// TIA Portal V19 program export: 4 tag tables, 0 data types, 0 data blocks, 3 code blocks (in call order from the OBs), 5 instance data blocks

VAR_GLOBAL   // PLC tag table "Alarm_Tags"
   ACKPB AT %M3.3 : Bool;   // Alarm ACK
   RESETPB AT %M3.4 : Bool;   // Alarm Reset
   Alarm_1 AT %M3.5 : Bool;   // Alarm #No1
   Alarm1ACKED AT %M3.6 : Bool;   // Alarm #1 Acknowledged
   Alarm1LED AT %M3.7 : Bool;   // Alarm #1 LED
   StopBelt AT %M4.0 : Bool;   // E-Stop The Belt
   Alarm_2 AT %M4.1 : Bool;   // Alarm #No2
   Alarm2ACKED AT %M4.2 : Bool;   // Alarm #2 Acknowledged
   Alarm2LED AT %M4.3 : Bool;   // Alarm #2 LED
END_VAR

VAR_GLOBAL   // PLC tag table "Clock_Tags"
   Clock_Byte AT %MB0 : Byte;
   Clock_10Hz AT %M0.0 : Bool;
   Clock_5Hz AT %M0.1 : Bool;
   "Clock_2.5Hz" AT %M0.2 : Bool;
   Clock_2Hz AT %M0.3 : Bool;
   "Clock_1.25Hz" AT %M0.4 : Bool;
   Clock_1Hz AT %M0.5 : Bool;
   "Clock_0.625Hz" AT %M0.6 : Bool;
   "Clock_0.5Hz" AT %M0.7 : Bool;
END_VAR

VAR_GLOBAL   // PLC tag table "Level_Tags"
   Pump1_Mode AT %M5.1 : Bool;   // Running Mode ( Auto or Manual)
   Pump1_Start_Manual AT %M5.2 : Bool;   // Start Manual Mode
   Pump1_Stop_Manual AT %M5.3 : Bool;   // Stop Manual Mode
   Pump1_Start_Auto AT %M5.4 : Bool;   // Start Auto Mode
   Pump1_Stop_Auto AT %M5.5 : Bool;   // Stop Auto Mode
   Level_High AT %M5.6 : Bool;   // High Level Reached
   Level_Low AT %M5.7 : Bool;   // Low Level Reached
   Timer_Setting_Run AT %MD6 : DInt;   // Timer Settings for Running
   Pump1_Overload AT %M10.0 : Bool;   // Pump Overloaded
   Pump1_Reset_Fault AT %M10.1 : Bool;   // Pump Reset Fault
   Pump1 AT %Q0.0 : Bool;   // Pump 1 - Output
   Pump1_Fault AT %M10.2 : Bool;   // Pump 1 Fault Status
   Pump1_Run_Auto_Activated AT %M10.3 : Bool;   // Pump 1 Running in Auto
   Level_Meter AT %MW12 : Int;   // Level Meter Reading
   Sensor_Real AT %QD2 : Real;   // Real Sensor Reading ( Tank Level)
   High_SP AT %MD14 : Real;   // High Setpoint
   Low_SP AT %MD18 : Real;   // Low Setpoint
END_VAR

VAR_GLOBAL   // PLC tag table "Mixer_Tags"
   Mixer_Start_PB AT %M4.5 : Bool;   // Starts Mixer
   Mixer_Stop_PB AT %M4.6 : Bool;   // Stops Mixer
   Mixer_Hold AT %M4.7 : Bool;   // Mixer held In Running
   Mixer AT %M5.0 : Bool;   // Mixer Status
   "2Hz_Mixer" AT %M4.4 : Bool;   // 2HZ Signal
END_VAR

ORGANIZATION_BLOCK "Main"   // OB1, LAD, ProgramCycle
TITLE = "Main Program Sweep (Cycle)"
{ S7_Optimized_Access := 'TRUE' }
// stored: SetENOAutomatically false
   VAR_INPUT
      Initial_Call : Bool;   // Initial call of this OB
      Remanence : Bool;   // =True, if remanent data are available
   END_VAR
BEGIN

REGION Network 1: Dispenser
   // Running Code - Dispenser Project
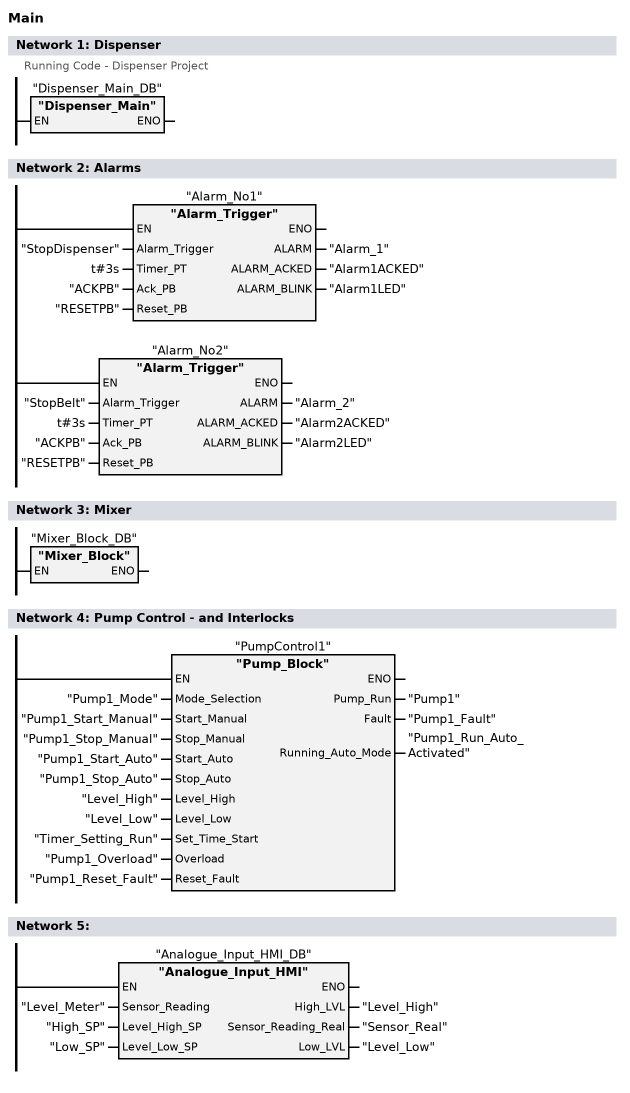
   RUNG wire#powerrail
      "Dispenser_Main_DB"()
   END_RUNG
   // the same network as SCL:
   "Dispenser_Main_DB"();   // "Dispenser_Main"
END_REGION

REGION Network 2: Alarms
   RUNG wire#powerrail
      "Alarm_No1"(Alarm_Trigger := "StopDispenser", Timer_PT := t#3s, Ack_PB := "ACKPB", Reset_PB := "RESETPB", ALARM => "Alarm_1", ALARM_ACKED => "Alarm1ACKED", ALARM_BLINK => "Alarm1LED")
   END_RUNG
   RUNG wire#powerrail
      "Alarm_No2"(Alarm_Trigger := "StopBelt", Timer_PT := t#3s, Ack_PB := "ACKPB", Reset_PB := "RESETPB", ALARM => "Alarm_2", ALARM_ACKED => "Alarm2ACKED", ALARM_BLINK => "Alarm2LED")
   END_RUNG
   // the same network as SCL:
   "Alarm_No1"(Alarm_Trigger := "StopDispenser",   // "Alarm_Trigger"
               Timer_PT := t#3s,
               Ack_PB := "ACKPB",
               Reset_PB := "RESETPB",
               ALARM => "Alarm_1",
               ALARM_ACKED => "Alarm1ACKED",
               ALARM_BLINK => "Alarm1LED");
   "Alarm_No2"(Alarm_Trigger := "StopBelt",   // "Alarm_Trigger"
               Timer_PT := t#3s,
               Ack_PB := "ACKPB",
               Reset_PB := "RESETPB",
               ALARM => "Alarm_2",
               ALARM_ACKED => "Alarm2ACKED",
               ALARM_BLINK => "Alarm2LED");
END_REGION

REGION Network 3: Mixer
   RUNG wire#powerrail
      "Mixer_Block_DB"()
   END_RUNG
   // the same network as SCL:
   "Mixer_Block_DB"();   // "Mixer_Block"
END_REGION

REGION Network 4: Pump Control - and Interlocks
   RUNG wire#powerrail
      "PumpControl1"(Mode_Selection := "Pump1_Mode", Start_Manual := "Pump1_Start_Manual", Stop_Manual := "Pump1_Stop_Manual", Start_Auto := "Pump1_Start_Auto", Stop_Auto := "Pump1_Stop_Auto", Level_High := "Level_High", Level_Low := "Level_Low", Set_Time_Start := "Timer_Setting_Run", Overload := "Pump1_Overload", Reset_Fault := "Pump1_Reset_Fault", Pump_Run => "Pump1", Fault => "Pump1_Fault", Running_Auto_Mode => "Pump1_Run_Auto_Activated")
   END_RUNG
   // the same network as SCL:
   "PumpControl1"(Mode_Selection := "Pump1_Mode",   // "Pump_Block"
                  Start_Manual := "Pump1_Start_Manual",
                  Stop_Manual := "Pump1_Stop_Manual",
                  Start_Auto := "Pump1_Start_Auto",
                  Stop_Auto := "Pump1_Stop_Auto",
                  Level_High := "Level_High",
                  Level_Low := "Level_Low",
                  Set_Time_Start := "Timer_Setting_Run",
                  Overload := "Pump1_Overload",
                  Reset_Fault := "Pump1_Reset_Fault",
                  Pump_Run => "Pump1",
                  Fault => "Pump1_Fault",
                  Running_Auto_Mode => "Pump1_Run_Auto_Activated");
END_REGION

REGION Network 5
   RUNG wire#powerrail
      "Analogue_Input_HMI_DB"(Sensor_Reading := "Level_Meter", Level_High_SP := "High_SP", Level_Low_SP := "Low_SP", High_LVL => "Level_High", Sensor_Reading_Real => "Sensor_Real", Low_LVL => "Level_Low")
   END_RUNG
   // the same network as SCL:
   "Analogue_Input_HMI_DB"(Sensor_Reading := "Level_Meter",   // "Analogue_Input_HMI"
                           Level_High_SP := "High_SP",
                           Level_Low_SP := "Low_SP",
                           High_LVL => "Level_High",
                           Sensor_Reading_Real => "Sensor_Real",
                           Low_LVL => "Level_Low");
END_REGION
END_ORGANIZATION_BLOCK

FUNCTION_BLOCK "Dispenser_Main"   // FB1, LAD
TITLE = Main Block for Dispenser Element and Conveyor Running
{ S7_Optimized_Access := 'TRUE' }
// Holds Code for Dispenser Project , Light Gates and Conveyor Belt Motor.
// stored: MemoryReserve 100, SetENOAutomatically false
   VAR_TEMP   // added for the SCL form of the ladder/FBD networks
      _w1 : Bool;
   END_VAR
BEGIN

REGION Network 1: Power Up
   // Enabled Power To System
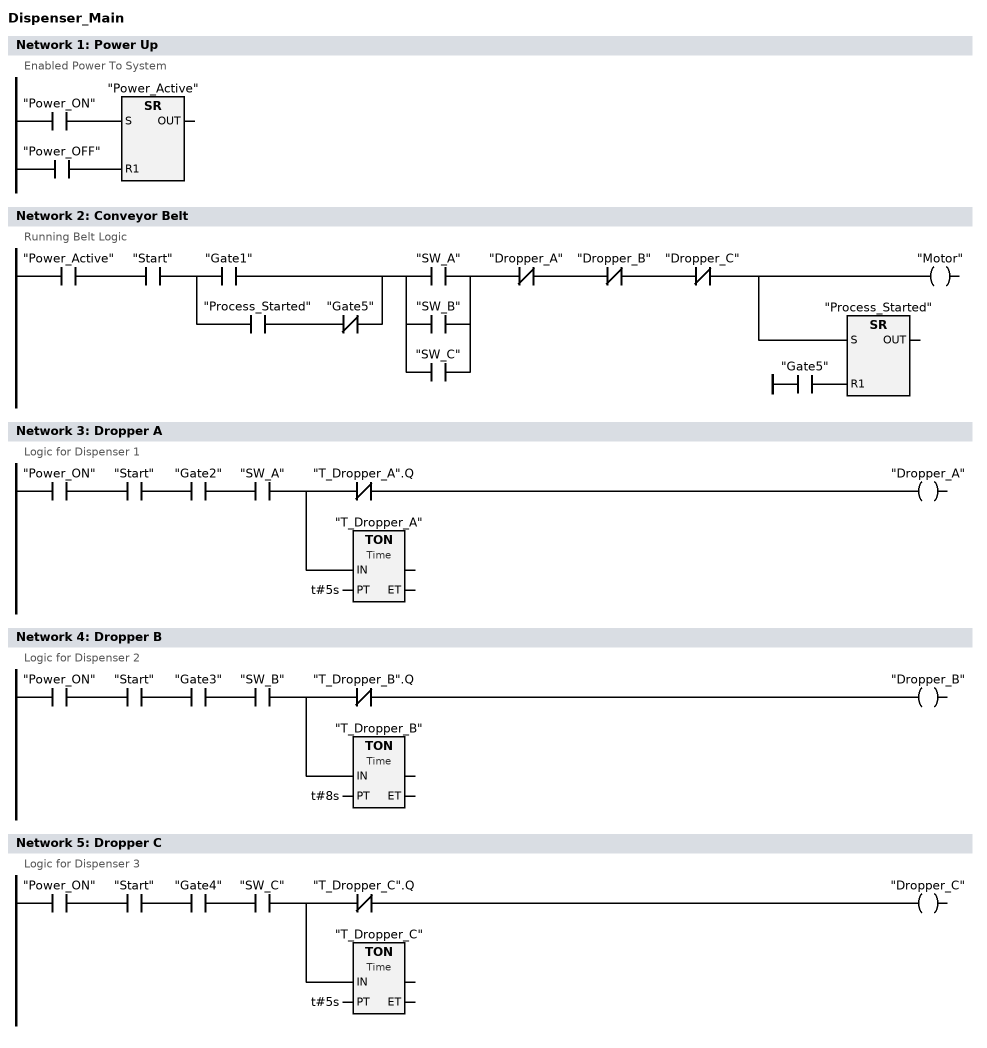
   RUNG wire#powerrail
      Contact( "Power_ON" )
      S_SR(operand := "Power_Active", r1 := wire#w1)
   END_RUNG
   RUNG wire#powerrail
      Contact( "Power_OFF" )
   END_RUNG wire#w1
   // the same network as SCL:
   IF "Power_ON" THEN
       "Power_Active" := TRUE;   // SR flip-flop
   END_IF;
   IF "Power_OFF" THEN "Power_Active" := FALSE; END_IF;
END_REGION

REGION Network 2: Conveyor Belt
   // Running Belt Logic
   RUNG wire#powerrail
      Contact( "Power_Active" )
      Contact( "Start" )
      wire#w1
      Contact( "Gate1" )
      wire#w2
      Contact( "SW_A" )
      wire#w3
      I_Contact( "Dropper_A" )
      I_Contact( "Dropper_B" )
      I_Contact( "Dropper_C" )
      wire#w4
      Coil( "Motor" )
   END_RUNG
   RUNG wire#w1
      Contact( "Process_Started" )
      I_Contact( "Gate5" )
   END_RUNG wire#w2
   RUNG wire#w2
      Contact( "SW_B" )
   END_RUNG wire#w3
   RUNG wire#w2
      Contact( "SW_C" )
   END_RUNG wire#w3
   RUNG wire#w4
      S_SR(operand := "Process_Started", r1 := wire#w5)
   END_RUNG
   RUNG wire#powerrail
      Contact( "Gate5" )
   END_RUNG wire#w5
   // the same network as SCL:
   "Motor" := "Power_Active" AND "Start" AND ("Gate1" OR ("Process_Started" AND NOT "Gate5")) AND ("SW_A" OR "SW_B" OR "SW_C") AND NOT "Dropper_A" AND NOT "Dropper_B" AND NOT "Dropper_C";
   IF "Motor" THEN
       "Process_Started" := TRUE;   // SR flip-flop
   END_IF;
   IF "Gate5" THEN "Process_Started" := FALSE; END_IF;
END_REGION

REGION Network 3: Dropper A
   // Logic for Dispenser 1
   RUNG wire#powerrail
      Contact( "Power_ON" )
      Contact( "Start" )
      Contact( "Gate2" )
      Contact( "SW_A" )
      wire#w1
      I_Contact( "T_Dropper_A".Q )
      Coil( "Dropper_A" )
   END_RUNG
   RUNG wire#w1
      { S7_Templates := "time_type := Time" } "T_Dropper_A".TON(pt := t#5s, et =>)
   END_RUNG
   // the same network as SCL:
   #_w1 := "Power_ON" AND "Start" AND "Gate2" AND "SW_A";
   "Dropper_A" := #_w1 AND NOT "T_Dropper_A".Q;
   "T_Dropper_A".TON(IN := #_w1, PT := t#5s);
END_REGION

REGION Network 4: Dropper B
   // Logic for Dispenser 2
   RUNG wire#powerrail
      Contact( "Power_ON" )
      Contact( "Start" )
      Contact( "Gate3" )
      Contact( "SW_B" )
      wire#w1
      I_Contact( "T_Dropper_B".Q )
      Coil( "Dropper_B" )
   END_RUNG
   RUNG wire#w1
      { S7_Templates := "time_type := Time" } "T_Dropper_B".TON(pt := t#8s, et =>)
   END_RUNG
   // the same network as SCL:
   #_w1 := "Power_ON" AND "Start" AND "Gate3" AND "SW_B";
   "Dropper_B" := #_w1 AND NOT "T_Dropper_B".Q;
   "T_Dropper_B".TON(IN := #_w1, PT := t#8s);
END_REGION

REGION Network 5: Dropper C
   // Logic for Dispenser 3
   RUNG wire#powerrail
      Contact( "Power_ON" )
      Contact( "Start" )
      Contact( "Gate4" )
      Contact( "SW_C" )
      wire#w1
      I_Contact( "T_Dropper_C".Q )
      Coil( "Dropper_C" )
   END_RUNG
   RUNG wire#w1
      { S7_Templates := "time_type := Time" } "T_Dropper_C".TON(pt := t#5s, et =>)
   END_RUNG
   // the same network as SCL:
   #_w1 := "Power_ON" AND "Start" AND "Gate4" AND "SW_C";
   "Dropper_C" := #_w1 AND NOT "T_Dropper_C".Q;
   "T_Dropper_C".TON(IN := #_w1, PT := t#5s);
END_REGION

REGION Network 6: Spare Network
END_REGION
END_FUNCTION_BLOCK

FUNCTION_BLOCK "Mixer_Block"   // FB3, LAD
TITLE = Control of Mixer Unit
{ S7_Optimized_Access := 'TRUE' }
// Simple Mixer Design and Animation
// stored: MemoryReserve 100, SetENOAutomatically false
BEGIN

REGION Network 1: Start Mixer
   // Turns Mixer On , Refreshes at 2Hz for Animation.
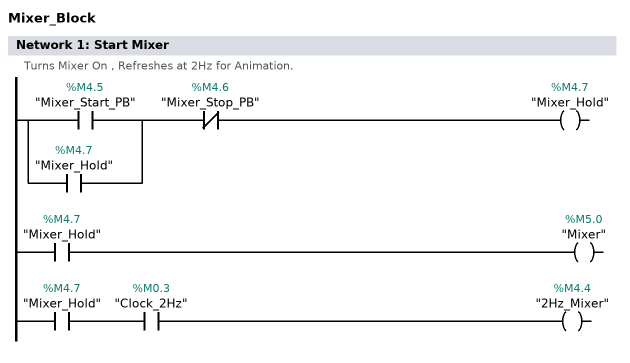
   RUNG wire#powerrail
      Contact( "Mixer_Start_PB" )
      wire#w1
      I_Contact( "Mixer_Stop_PB" )
      Coil( "Mixer_Hold" )
   END_RUNG
   RUNG wire#powerrail
      Contact( "Mixer_Hold" )
   END_RUNG wire#w1
   RUNG wire#powerrail
      Contact( "Mixer_Hold" )
      Coil( "Mixer" )
   END_RUNG
   RUNG wire#powerrail
      Contact( "Mixer_Hold" )
      Contact( "Clock_2Hz" )
      Coil( "2Hz_Mixer" )
   END_RUNG
   // the same network as SCL:
   "Mixer_Hold" := ("Mixer_Start_PB" OR "Mixer_Hold") AND NOT "Mixer_Stop_PB";
   "Mixer" := "Mixer_Hold";
   "2Hz_Mixer" := "Mixer_Hold" AND "Clock_2Hz";
END_REGION
END_FUNCTION_BLOCK

DATA_BLOCK "Alarm_No2"   // DB7
// stored: InstanceOfName Alarm_Trigger, InstanceOfType FB
"Alarm_Trigger"
   // VAR_INPUT
   //    Alarm_Trigger : Bool;
   //    Timer_PT : Time;
   //    Ack_PB : Bool;
   //    Reset_PB : Bool;
   // END_VAR
   // VAR_OUTPUT
   //    ALARM : Bool;
   //    ALARM_ACKED : Bool;
   //    ALARM_BLINK : Bool;
   // END_VAR
   // VAR
   //    Alarm_TD : Bool;
   //    Alarm_Active : Bool;
   //    Alarm_ACK : Bool;
   //    Alarm_Reset : Bool;
   //    Alarm_Timer { S7_SetPoint := 'True'} : TON_TIME;
   // END_VAR
BEGIN
END_DATA_BLOCK

DATA_BLOCK "Analogue_Input_HMI_DB"   // DB10
// stored: InstanceOfName Analogue_Input_HMI, InstanceOfType FB
"Analogue_Input_HMI"
   // VAR_INPUT
   //    Sensor_Reading { ExternalAccessible := 'False'; ExternalVisible := 'False'; ExternalWritable := 'False'} : Int;
   // END_VAR
   // VAR_OUTPUT
   //    High_LVL { ExternalAccessible := 'False'; ExternalVisible := 'False'; ExternalWritable := 'False'} : Bool;
   //    Sensor_Reading_Real { ExternalAccessible := 'False'; ExternalVisible := 'False'; ExternalWritable := 'False'} : Real;
   //    Low_LVL { ExternalAccessible := 'False'; ExternalVisible := 'False'; ExternalWritable := 'False'} : Bool;
   // END_VAR
   // VAR_IN_OUT
   //    Level_High_SP { ExternalAccessible := 'False'; ExternalVisible := 'False'; ExternalWritable := 'False'} : Real;
   //    Level_Low_SP { ExternalAccessible := 'False'; ExternalVisible := 'False'; ExternalWritable := 'False'} : Real;
   // END_VAR
BEGIN
END_DATA_BLOCK

DATA_BLOCK "Dispenser_Main_DB"   // DB4
// stored: InstanceOfName Dispenser_Main, InstanceOfType FB
"Dispenser_Main"
BEGIN
END_DATA_BLOCK

DATA_BLOCK "PumpControl1"   // DB9
// stored: InstanceOfName Pump_Block, InstanceOfType FB
"Pump_Block"
   // VAR_INPUT
   //    Mode_Selection : Bool;
   //    Start_Manual : Bool;
   //    Stop_Manual : Bool;
   //    Start_Auto : Bool;
   //    Stop_Auto : Bool;
   //    Level_High : Bool;
   //    Level_Low : Bool;
   //    Set_Time_Start : DInt;
   //    Overload : Bool;
   //    Reset_Fault : Bool;
   // END_VAR
   // VAR_OUTPUT
   //    Pump_Run : Bool;
   //    Fault : Bool;
   //    Running_Auto_Mode : Bool;
   // END_VAR
   // VAR
   //    Timer_Start : IEC_TIMER;
   //    Start_Auto_Activated : Bool;
   // END_VAR
BEGIN
END_DATA_BLOCK

DATA_BLOCK "Timer_Start"   // DB8
{ S7_Optimized_Access := 'TRUE' }
// stored: InstanceOfName IEC_TIMER, OfSystemLibElement IEC_TIMER, OfSystemLibVersion 1.0
"IEC_TIMER"
   // VAR
   //    PT : Time;
   //    ET { ExternalWritable := 'False'} : Time;
   //    IN : Bool;
   //    Q { ExternalWritable := 'False'} : Bool;
   // END_VAR
BEGIN
END_DATA_BLOCK
